TEXTLIST EL1904_M_3
  1 = 'interlock_out_cover' | chinese: 'OUT_透明盖' | Chinese: 'OUT_透明盖'
  2 = 'interlock_out_cover' | chinese: 'OUT_透明盖' | Chinese: 'OUT_透明盖'
  3 = 'interlock_out_left_door' | chinese: 'OUT_左侧上下门' | Chinese: 'OUT_左侧上下门'
  4 = 'interlock_out_left_door' | chinese: 'OUT_左侧上下门' | Chinese: 'OUT_左侧上下门'
   = ''
END_TEXTLIST

(* stored: Version 1.1.0.1, ProductVersion 3.1.4024.11
   TextList EL1904_M_3: Id {5f4b0639-f57e-4bc5-b60f-808c74be80a0} *)
